TYPE ST_DomeCharmber :
STRUCT
END_STRUCT
END_TYPE

(* stored: Version 1.1.0.1, ProductVersion 3.1.4024.12
   DUT ST_DomeCharmber: Id {7ab9f2cd-b9e4-4fab-bb2b-88192881c7fe} *)
